(* Logix 5000 project; controller cal1615 1756-L62 rev 20.19; software revision 20.05; part 53 of 82 *)
(* tags used below, declared in another part *)
   p23r17 : routine;
   FAULT : BOOL;   // Fault AFI
   HMI : BOOL;   // AFI HMI
   p01_param_oven_timer_presets : DINT[32];   // System Parameter Oven Timer Presets
   p01r09 : routine;   // System Modes
   p01r09_pb_global_reset : BOOL;   // System Modes PB: Global Fault Reset
   p01r11 : routine;   // System Timer Presets
   p01r13_line_running : BOOL;   // System Line Start Sequence Line Running
   p02_dint_from_hmi : hmi_dint;
   p02_real_from_hmi : hmi_real;   // MOP HMI Iface Real from HMI
   p23_ai_os_masked_gap : REAL;
   p23_ao_servo_os_zero_offset : REAL;   // Impreg Analog Outputs Drive Operator Side Servo Position Offset
   p23_di_servo_os : servo_di;   // Impreg Digital Inputs Servo Operator Side
   p23_di_vfd_jog_fwd : BOOL;   // Impreg Input PB: VFD Jog FWD
   p23_di_vfd_jog_rev : BOOL;   // Impreg Input PB: VFD Jog REV
   p23_dint_to_hmi : DINT[17];   // Impreg Dint to HMI
   p23_do_servo_os : servo_do;   // Impreg Digital Outputs Operator Side Servo
   p23_param_lfl_hhl : REAL;   // Impreg Parameter LFL High High Limit
   p23_param_lfl_hl : REAL;   // Impreg Parameters LFL High Limit
   p23_param_servo_open_position : REAL;
   p23_param_zone_pressure : REAL;   // MOP HMI Iface Parameters Minimum Pressure
   p23r01 : routine;   // Impreg Main
   p23r02 : routine;   // Impreg Misc Control
   p23r08 : routine;   // Impreg Warnings
   p23r08_timer_fault : TIMER[4];   // Impreg Warnings Fault Delay
   p23r08_timer_warning : TIMER[4];   // Impreg Warnings Warning Delay
   p23r09 : routine;   // Impreg Mode Selection
   p23r09_mode_run : BOOL;   // Impreg Modes Pick Up Roll Run Mode
   p23r09_timer_fault : TIMER[4];   // Impreg Mode Selection Fault Delay
   p23r09_web_wet_ctrl_toggle : SYS_Toggle;   // Impreg Metering Roll VFD Web Wet Control
   p23r10 : routine;
   p23r10_timer_fault : TIMER[4];   // Impreg Parameters Fault Dwell Timer
   p23r10_timer_warning : TIMER[4];   // Impreg Parameters Warning Dwell Timer
   p23r11 : routine;   // Impreg Servo Operator Side
   p23r11_gap_sequence_enabled : BOOL;
   p23r11_impreg_gap_os : REAL;
   p23r11_offsets : REAL[100];
   p23r11_permissive_jog : BOOL;   // Impreg Servo Operator Side Perimssive Jog
   p23r11_pos_offset : REAL;
   p23r11_request_jog_fwd : BOOL;   // Impreg Servo Operator Side Requset Jog Forward
   p23r11_request_jog_rev : BOOL;   // Impreg Servo Operator Side Requset Jog Reverse
   p23r11_request_position : BOOL;   // Impreg Servo Operator Side Request Position
   p23r11_request_start : BOOL;   // Impreg Servo Operator Side Request Start
   p23r11_request_zero : BOOL;   // Impreg Servo Operator Side Request Zero
   p23r11_selected_position : REAL;
   p23r11_servo_not_ready : BOOL;   // Impreg Servo Operator Side Not Ready
   p23r11_servo_status_ab : BOOL;   // Impreg Servo Operator Side AB Status
   p23r11_servo_status_af : BOOL;   // Impreg Servo Operator Side AF Status
   p23r11_servo_status_bb : BOOL;   // Impreg Servo Operator Side BB Status
   p23r11_step_4_dwell : TIMER;
   p23r11_timer : TIMER[4];   // Impreg Servo Operator Side Timer
   p23r12 : routine;   // Impreg Servo Drive Side
   p23r13 : routine;
   p23r15 : routine;   // Impreg Metering Roll VFD
   p23r15_pid_tension_control : BOOL;   // Impreg Metering Roll VFD PID Wet Web Active
(* P23_Impreg, continued *)

ROUTINE R08_Warnings   (* ladder *)
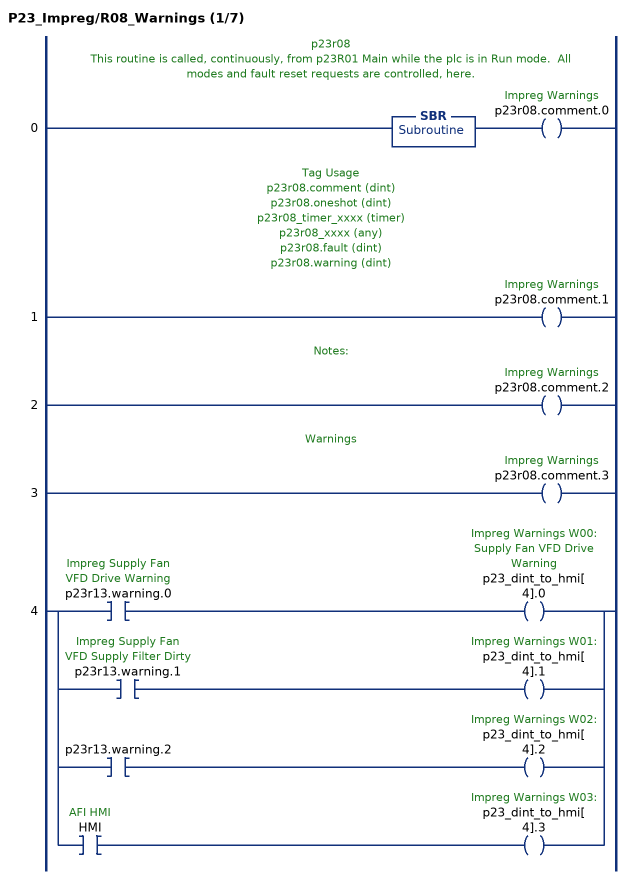
   // p23r08
   // This routine is called, continuously, from p23R01 Main while the plc is in Run mode.  All modes and fault reset requests are controlled, here.
   0: SBR()OTE(p23r08.comment.0);
   // Tag Usage
   // p23r08.comment (dint)
   // p23r08.oneshot (dint)
   // p23r08_timer_xxxx (timer)
   // p23r08_xxxx (any)
   // p23r08.fault (dint)
   // p23r08.warning (dint)
   1: OTE(p23r08.comment.1);
   // Notes:
   2: OTE(p23r08.comment.2);
   // Warnings
   3: OTE(p23r08.comment.3);
   4: [XIC(p23r13.warning.0) OTE(p23_dint_to_hmi[4].0) ,XIC(p23r13.warning.1) OTE(p23_dint_to_hmi[4].1) ,XIC(p23r13.warning.2) OTE(p23_dint_to_hmi[4].2) ,XIC(HMI) OTE(p23_dint_to_hmi[4].3) ];
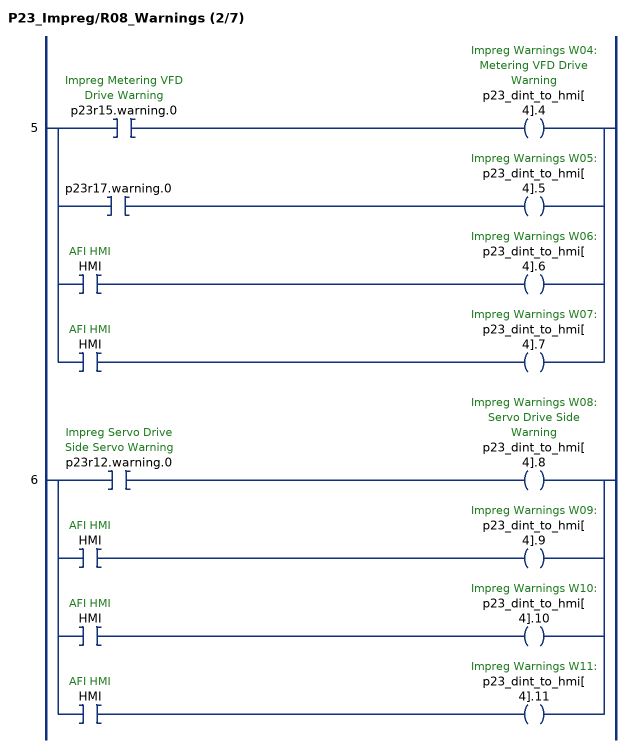
   5: [XIC(p23r15.warning.0) OTE(p23_dint_to_hmi[4].4) ,XIC(p23r17.warning.0) OTE(p23_dint_to_hmi[4].5) ,XIC(HMI) OTE(p23_dint_to_hmi[4].6) ,XIC(HMI) OTE(p23_dint_to_hmi[4].7) ];
   6: [XIC(p23r12.warning.0) OTE(p23_dint_to_hmi[4].8) ,XIC(HMI) OTE(p23_dint_to_hmi[4].9) ,XIC(HMI) OTE(p23_dint_to_hmi[4].10) ,XIC(HMI) OTE(p23_dint_to_hmi[4].11) ];
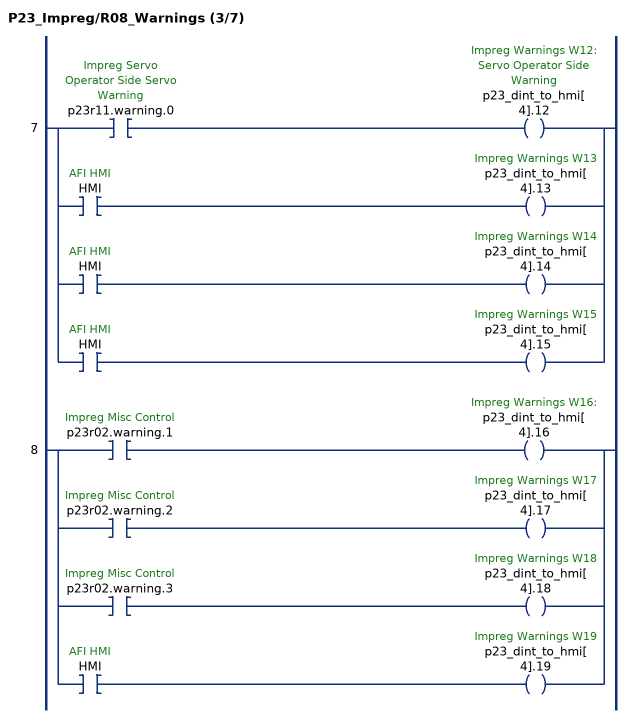
   7: [XIC(p23r11.warning.0) OTE(p23_dint_to_hmi[4].12) ,XIC(HMI) OTE(p23_dint_to_hmi[4].13) ,XIC(HMI) OTE(p23_dint_to_hmi[4].14) ,XIC(HMI) OTE(p23_dint_to_hmi[4].15) ];
   8: [XIC(p23r02.warning.1) OTE(p23_dint_to_hmi[4].16) ,XIC(p23r02.warning.2) OTE(p23_dint_to_hmi[4].17) ,XIC(p23r02.warning.3) OTE(p23_dint_to_hmi[4].18) ,XIC(HMI) OTE(p23_dint_to_hmi[4].19) ];
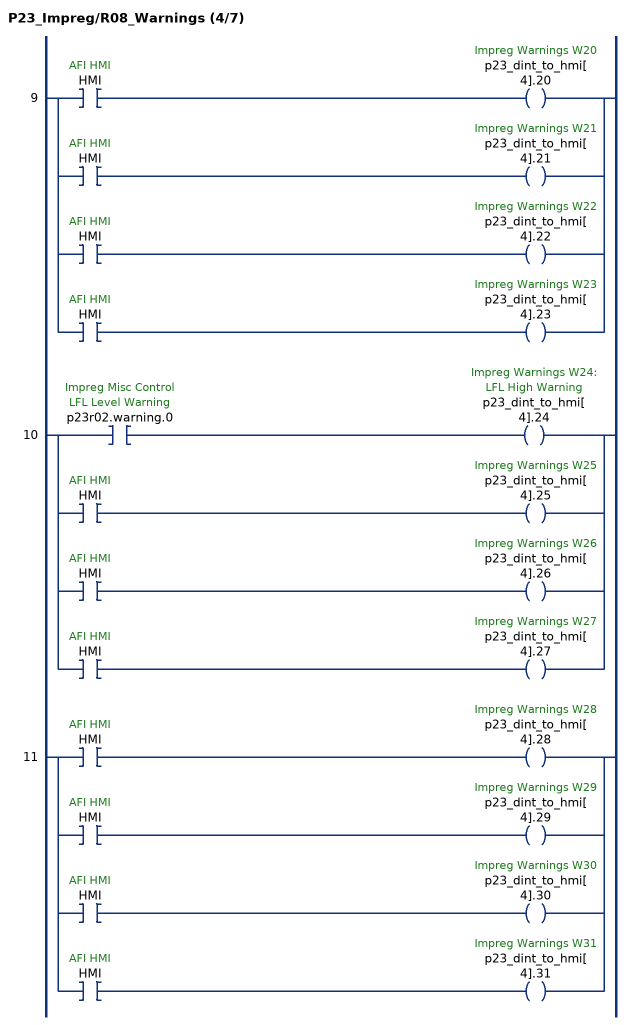
   9: [XIC(HMI) OTE(p23_dint_to_hmi[4].20) ,XIC(HMI) OTE(p23_dint_to_hmi[4].21) ,XIC(HMI) OTE(p23_dint_to_hmi[4].22) ,XIC(HMI) OTE(p23_dint_to_hmi[4].23) ];
   10: [XIC(p23r02.warning.0) OTE(p23_dint_to_hmi[4].24) ,XIC(HMI) OTE(p23_dint_to_hmi[4].25) ,XIC(HMI) OTE(p23_dint_to_hmi[4].26) ,XIC(HMI) OTE(p23_dint_to_hmi[4].27) ];
   11: [XIC(HMI) OTE(p23_dint_to_hmi[4].28) ,XIC(HMI) OTE(p23_dint_to_hmi[4].29) ,XIC(HMI) OTE(p23_dint_to_hmi[4].30) ,XIC(HMI) OTE(p23_dint_to_hmi[4].31) ];
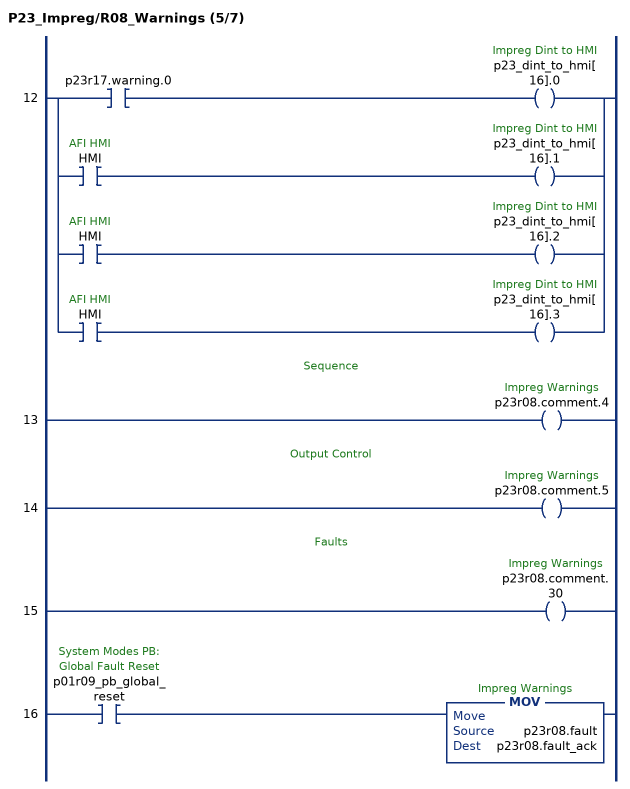
   12: [XIC(p23r17.warning.0) OTE(p23_dint_to_hmi[16].0) ,XIC(HMI) OTE(p23_dint_to_hmi[16].1) ,XIC(HMI) OTE(p23_dint_to_hmi[16].2) ,XIC(HMI) OTE(p23_dint_to_hmi[16].3) ];
   // Sequence
   13: OTE(p23r08.comment.4);
   // Output Control
   14: OTE(p23r08.comment.5);
   // Faults
   15: OTE(p23r08.comment.30);
   16: XIC(p01r09_pb_global_reset)MOV(p23r08.fault,p23r08.fault_ack);
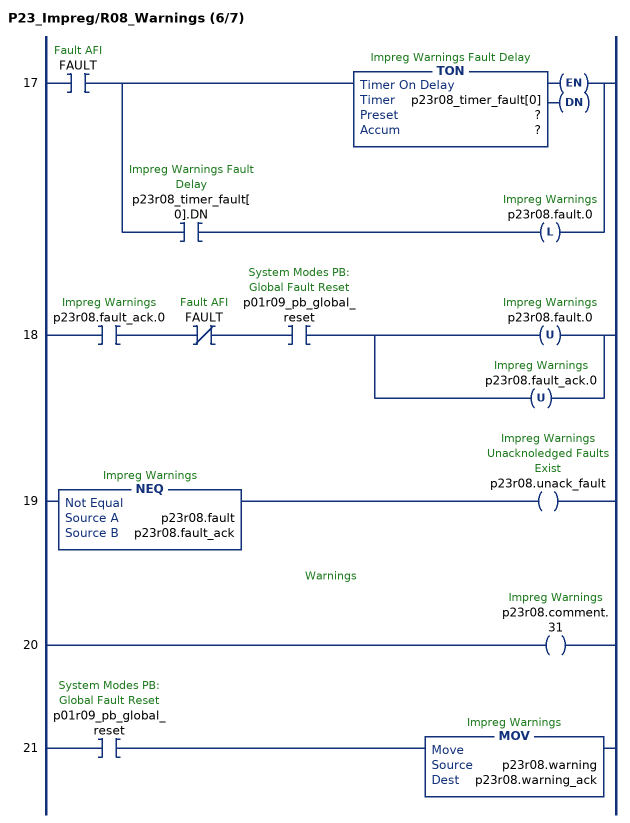
   17: XIC(FAULT)[TON(p23r08_timer_fault[0],?,?) ,XIC(p23r08_timer_fault[0].DN) OTL(p23r08.fault.0) ];
   18: XIC(p23r08.fault_ack.0)XIO(FAULT)XIC(p01r09_pb_global_reset)[OTU(p23r08.fault.0) ,OTU(p23r08.fault_ack.0) ];
   19: NEQ(p23r08.fault,p23r08.fault_ack)OTE(p23r08.unack_fault);
   // Warnings
   20: OTE(p23r08.comment.31);
   21: XIC(p01r09_pb_global_reset)MOV(p23r08.warning,p23r08.warning_ack);
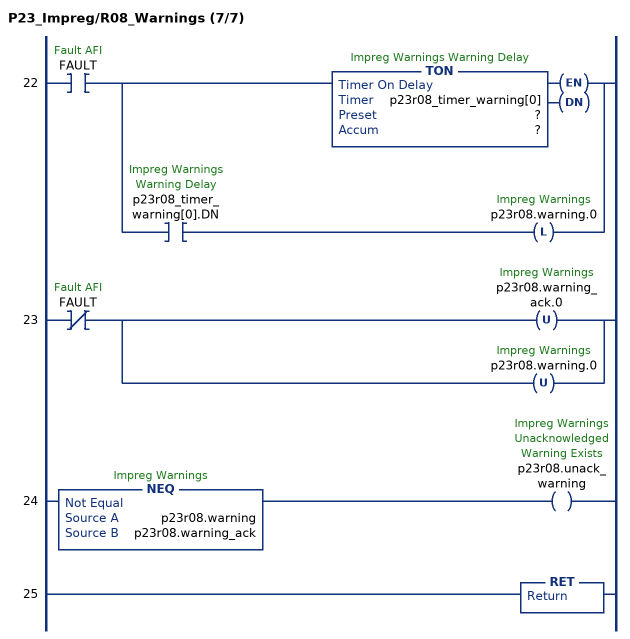
   22: XIC(FAULT)[TON(p23r08_timer_warning[0],?,?) ,XIC(p23r08_timer_warning[0].DN) OTL(p23r08.warning.0) ];
   23: XIO(FAULT)[OTU(p23r08.warning_ack.0) ,OTU(p23r08.warning.0) ];
   24: NEQ(p23r08.warning,p23r08.warning_ack)OTE(p23r08.unack_warning);
   25: RET();
END_ROUTINE

ROUTINE R09_Modes   (* ladder *)
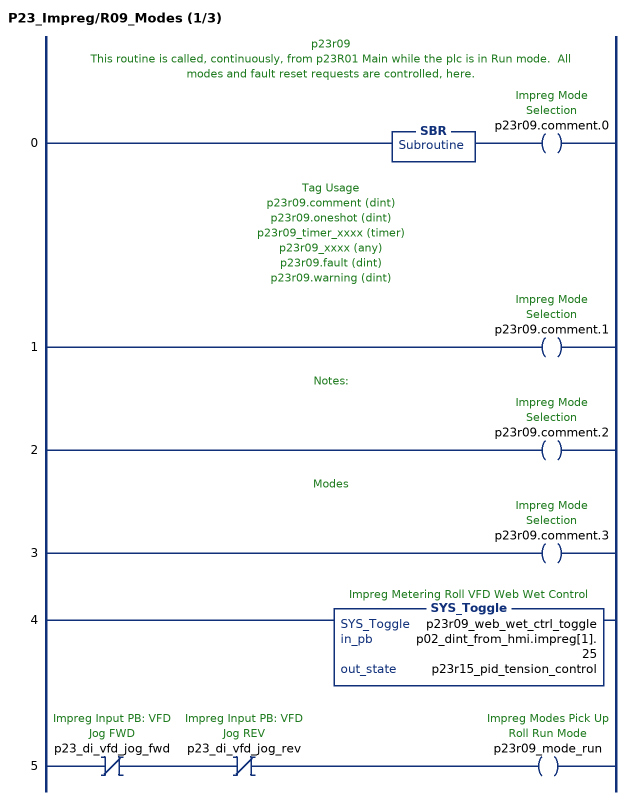
   // p23r09
   // This routine is called, continuously, from p23R01 Main while the plc is in Run mode.  All modes and fault reset requests are controlled, here.
   0: SBR()OTE(p23r09.comment.0);
   // Tag Usage
   // p23r09.comment (dint)
   // p23r09.oneshot (dint)
   // p23r09_timer_xxxx (timer)
   // p23r09_xxxx (any)
   // p23r09.fault (dint)
   // p23r09.warning (dint)
   1: OTE(p23r09.comment.1);
   // Notes:
   2: OTE(p23r09.comment.2);
   // Modes
   3: OTE(p23r09.comment.3);
   4: SYS_Toggle(p23r09_web_wet_ctrl_toggle,p02_dint_from_hmi.impreg[1].25,p23r15_pid_tension_control);
   5: XIO(p23_di_vfd_jog_fwd)XIO(p23_di_vfd_jog_rev)OTE(p23r09_mode_run);
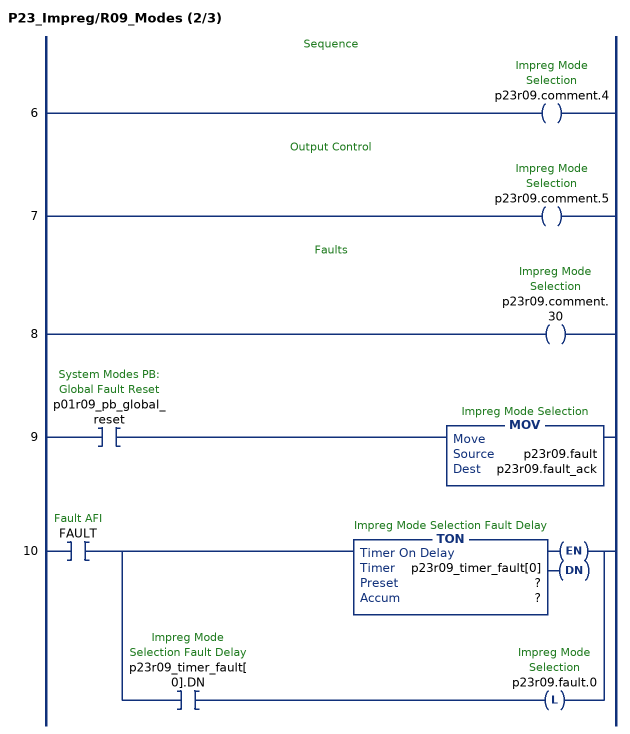
   // Sequence
   6: OTE(p23r09.comment.4);
   // Output Control
   7: OTE(p23r09.comment.5);
   // Faults
   8: OTE(p23r09.comment.30);
   9: XIC(p01r09_pb_global_reset)MOV(p23r09.fault,p23r09.fault_ack);
   10: XIC(FAULT)[TON(p23r09_timer_fault[0],?,?) ,XIC(p23r09_timer_fault[0].DN) OTL(p23r09.fault.0) ];
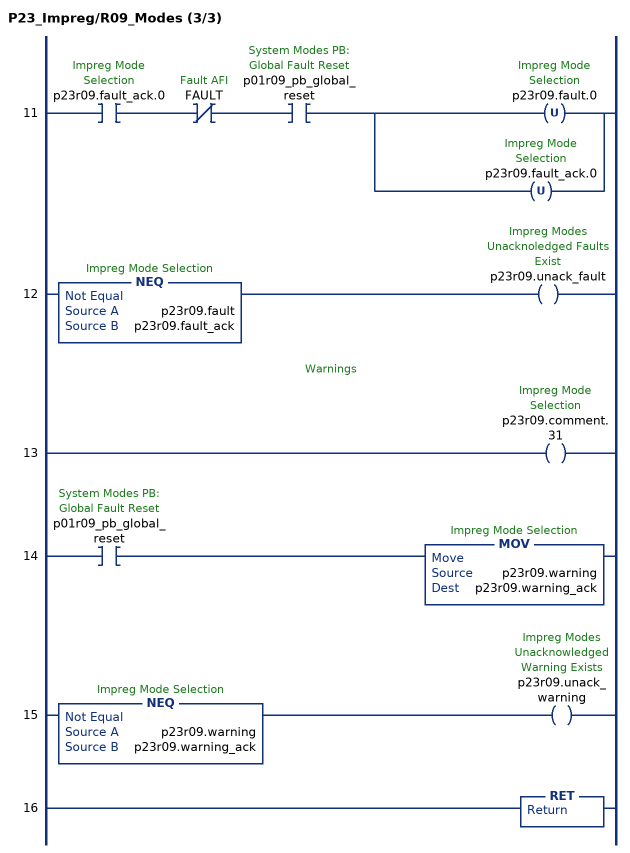
   11: XIC(p23r09.fault_ack.0)XIO(FAULT)XIC(p01r09_pb_global_reset)[OTU(p23r09.fault.0) ,OTU(p23r09.fault_ack.0) ];
   12: NEQ(p23r09.fault,p23r09.fault_ack)OTE(p23r09.unack_fault);
   // Warnings
   13: OTE(p23r09.comment.31);
   14: XIC(p01r09_pb_global_reset)MOV(p23r09.warning,p23r09.warning_ack);
   15: NEQ(p23r09.warning,p23r09.warning_ack)OTE(p23r09.unack_warning);
   16: RET();
END_ROUTINE

ROUTINE R10_Parameters   (* ladder *)
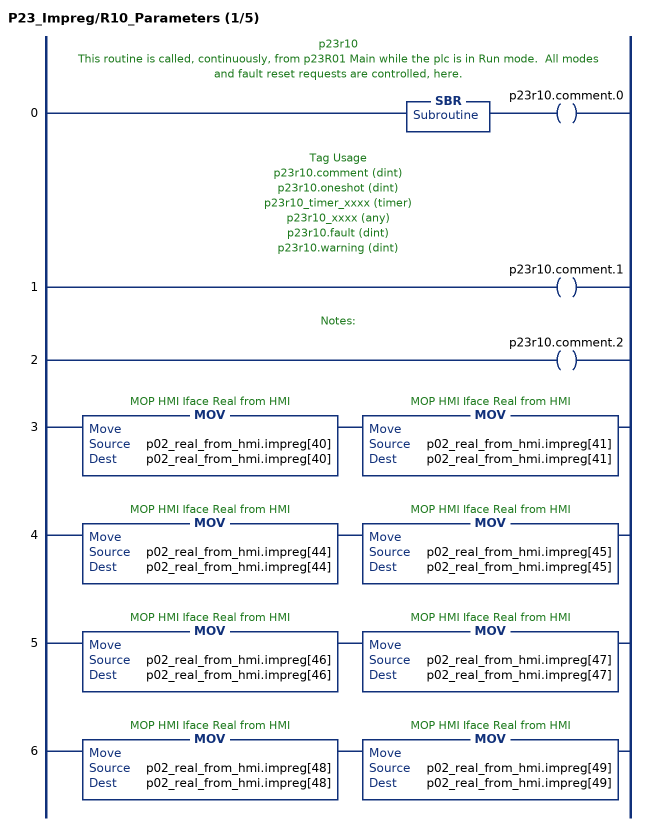
   // p23r10
   // This routine is called, continuously, from p23R01 Main while the plc is in Run mode.  All modes and fault reset requests are controlled, here.
   0: SBR()OTE(p23r10.comment.0);
   // Tag Usage
   // p23r10.comment (dint)
   // p23r10.oneshot (dint)
   // p23r10_timer_xxxx (timer)
   // p23r10_xxxx (any)
   // p23r10.fault (dint)
   // p23r10.warning (dint)
   1: OTE(p23r10.comment.1);
   // Notes:
   2: OTE(p23r10.comment.2);
   3: MOV(p02_real_from_hmi.impreg[40],p02_real_from_hmi.impreg[40])MOV(p02_real_from_hmi.impreg[41],p02_real_from_hmi.impreg[41]);
   4: MOV(p02_real_from_hmi.impreg[44],p02_real_from_hmi.impreg[44])MOV(p02_real_from_hmi.impreg[45],p02_real_from_hmi.impreg[45]);
   5: MOV(p02_real_from_hmi.impreg[46],p02_real_from_hmi.impreg[46])MOV(p02_real_from_hmi.impreg[47],p02_real_from_hmi.impreg[47]);
   6: MOV(p02_real_from_hmi.impreg[48],p02_real_from_hmi.impreg[48])MOV(p02_real_from_hmi.impreg[49],p02_real_from_hmi.impreg[49]);
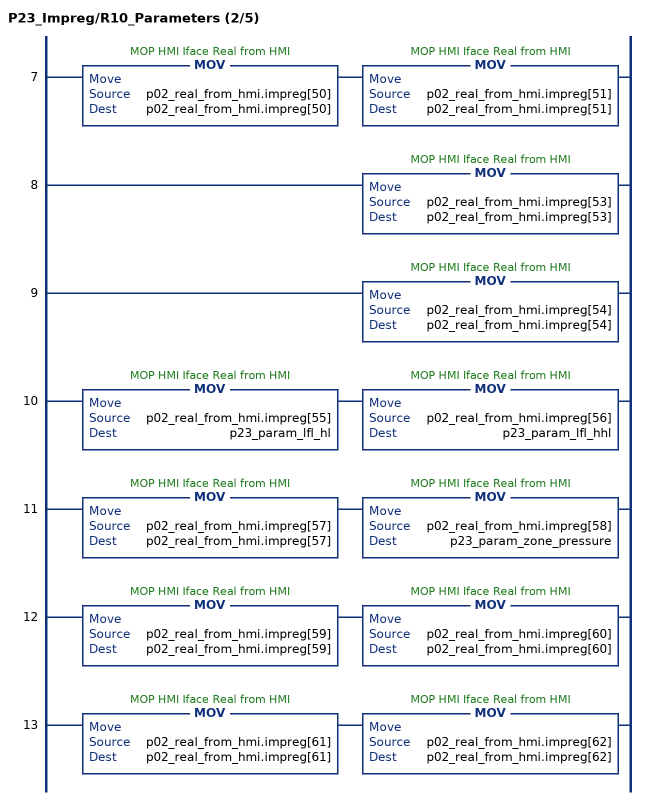
   7: MOV(p02_real_from_hmi.impreg[50],p02_real_from_hmi.impreg[50])MOV(p02_real_from_hmi.impreg[51],p02_real_from_hmi.impreg[51]);
   8: MOV(p02_real_from_hmi.impreg[53],p02_real_from_hmi.impreg[53]);
   9: MOV(p02_real_from_hmi.impreg[54],p02_real_from_hmi.impreg[54]);
   10: MOV(p02_real_from_hmi.impreg[55],p23_param_lfl_hl)MOV(p02_real_from_hmi.impreg[56],p23_param_lfl_hhl);
   11: MOV(p02_real_from_hmi.impreg[57],p02_real_from_hmi.impreg[57])MOV(p02_real_from_hmi.impreg[58],p23_param_zone_pressure);
   12: MOV(p02_real_from_hmi.impreg[59],p02_real_from_hmi.impreg[59])MOV(p02_real_from_hmi.impreg[60],p02_real_from_hmi.impreg[60]);
   13: MOV(p02_real_from_hmi.impreg[61],p02_real_from_hmi.impreg[61])MOV(p02_real_from_hmi.impreg[62],p02_real_from_hmi.impreg[62]);
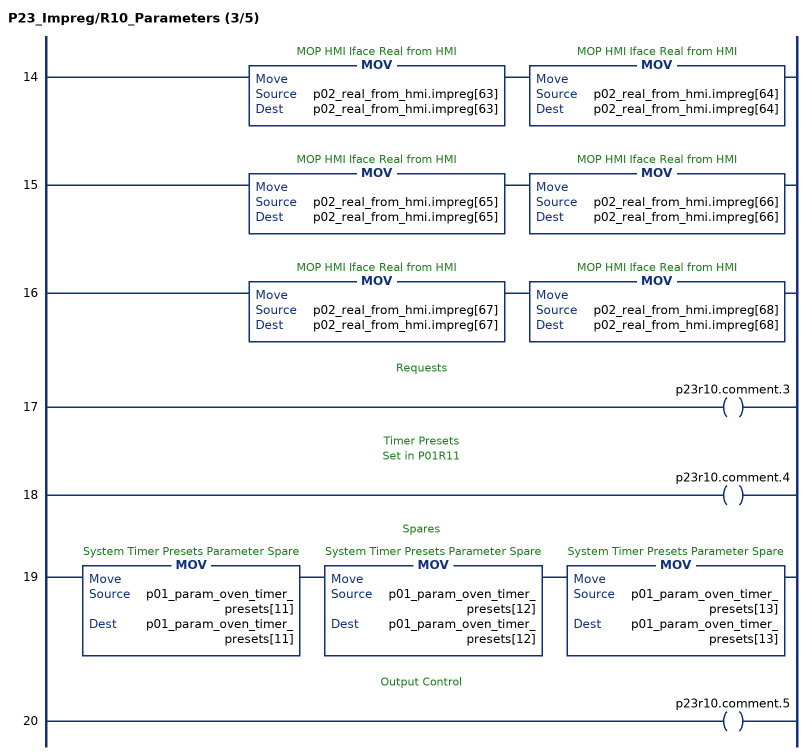
   14: MOV(p02_real_from_hmi.impreg[63],p02_real_from_hmi.impreg[63])MOV(p02_real_from_hmi.impreg[64],p02_real_from_hmi.impreg[64]);
   15: MOV(p02_real_from_hmi.impreg[65],p02_real_from_hmi.impreg[65])MOV(p02_real_from_hmi.impreg[66],p02_real_from_hmi.impreg[66]);
   16: MOV(p02_real_from_hmi.impreg[67],p02_real_from_hmi.impreg[67])MOV(p02_real_from_hmi.impreg[68],p02_real_from_hmi.impreg[68]);
   // Requests
   17: OTE(p23r10.comment.3);
   // Timer Presets
   // Set in P01R11
   18: OTE(p23r10.comment.4);
   // Spares
   19: MOV(p01_param_oven_timer_presets[11],p01_param_oven_timer_presets[11])MOV(p01_param_oven_timer_presets[12],p01_param_oven_timer_presets[12])MOV(p01_param_oven_timer_presets[13],p01_param_oven_timer_presets[13]);
   // Output Control
   20: OTE(p23r10.comment.5);
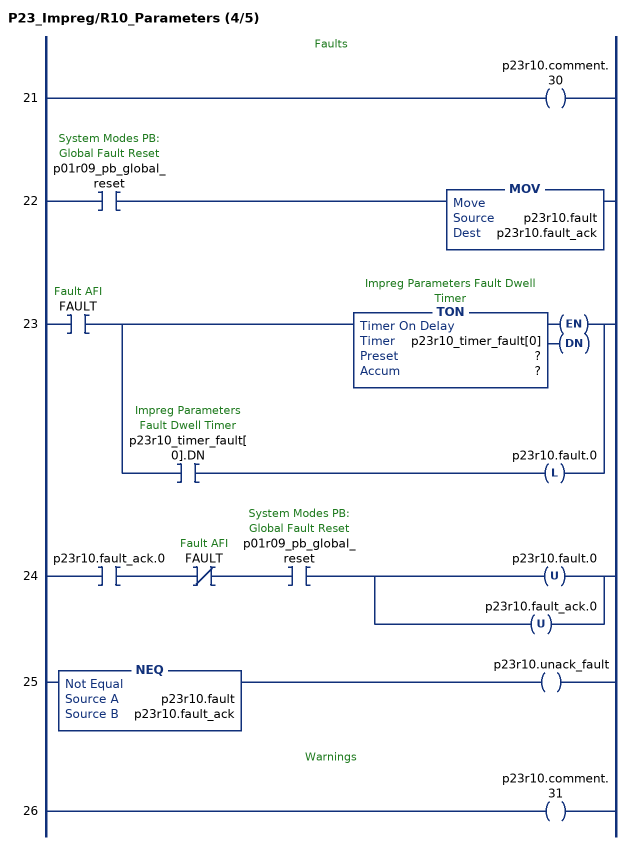
   // Faults
   21: OTE(p23r10.comment.30);
   22: XIC(p01r09_pb_global_reset)MOV(p23r10.fault,p23r10.fault_ack);
   23: XIC(FAULT)[TON(p23r10_timer_fault[0],?,?) ,XIC(p23r10_timer_fault[0].DN) OTL(p23r10.fault.0) ];
   24: XIC(p23r10.fault_ack.0)XIO(FAULT)XIC(p01r09_pb_global_reset)[OTU(p23r10.fault.0) ,OTU(p23r10.fault_ack.0) ];
   25: NEQ(p23r10.fault,p23r10.fault_ack)OTE(p23r10.unack_fault);
   // Warnings
   26: OTE(p23r10.comment.31);
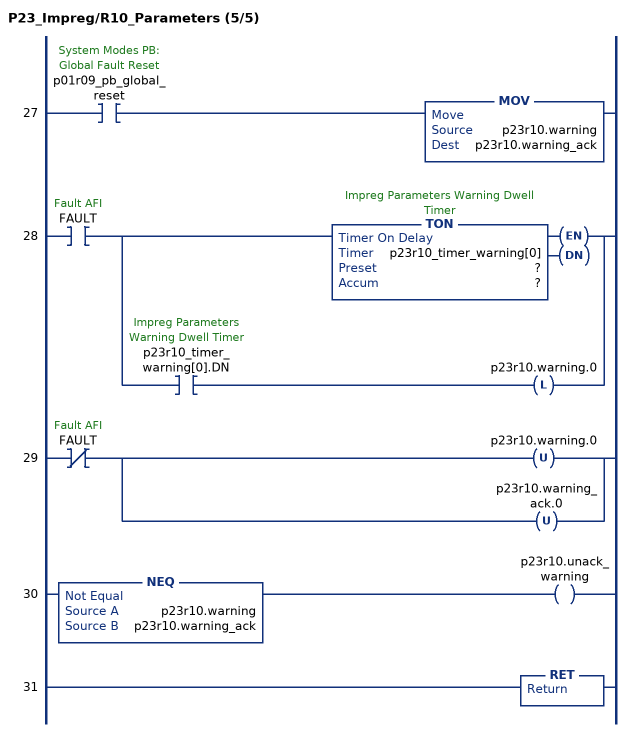
   27: XIC(p01r09_pb_global_reset)MOV(p23r10.warning,p23r10.warning_ack);
   28: XIC(FAULT)[TON(p23r10_timer_warning[0],?,?) ,XIC(p23r10_timer_warning[0].DN) OTL(p23r10.warning.0) ];
   29: XIO(FAULT)[OTU(p23r10.warning.0) ,OTU(p23r10.warning_ack.0) ];
   30: NEQ(p23r10.warning,p23r10.warning_ack)OTE(p23r10.unack_warning);
   31: RET();
END_ROUTINE

ROUTINE R11_Servo_Operator_Side   (* ladder *)
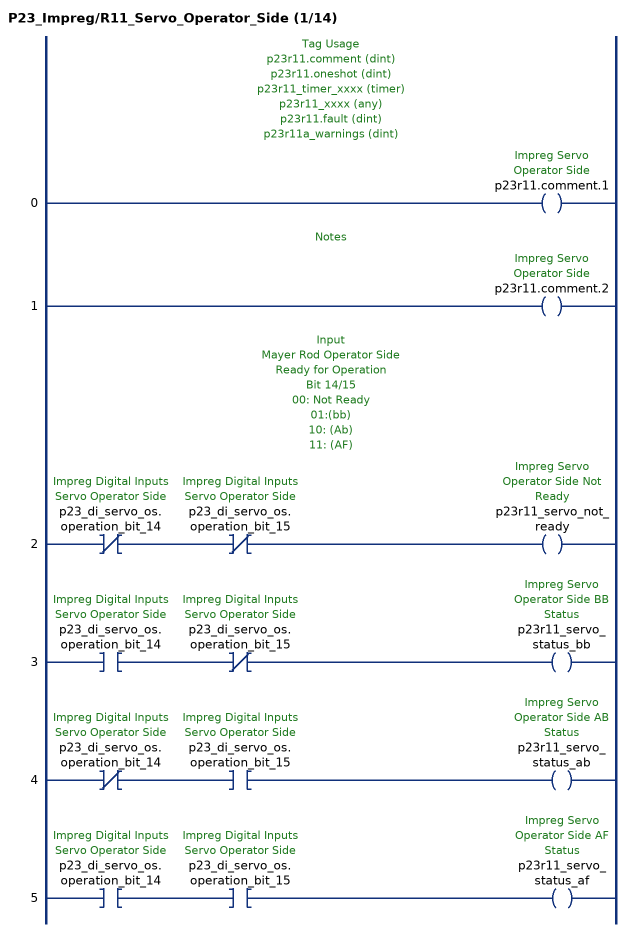
   // Tag Usage
   // p23r11.comment (dint)
   // p23r11.oneshot (dint)
   // p23r11_timer_xxxx (timer)
   // p23r11_xxxx (any)
   // p23r11.fault (dint)
   // p23r11a_warnings (dint)
   0: OTE(p23r11.comment.1);
   // Notes
   1: OTE(p23r11.comment.2);
   // Input
   // Mayer Rod Operator Side
   // Ready for Operation
   // Bit 14/15
   // 00: Not Ready
   // 01:(bb)
   // 10: (Ab)
   // 11: (AF)
   2: XIO(p23_di_servo_os.operation_bit_14)XIO(p23_di_servo_os.operation_bit_15)OTE(p23r11_servo_not_ready);
   3: XIC(p23_di_servo_os.operation_bit_14)XIO(p23_di_servo_os.operation_bit_15)OTE(p23r11_servo_status_bb);
   4: XIO(p23_di_servo_os.operation_bit_14)XIC(p23_di_servo_os.operation_bit_15)OTE(p23r11_servo_status_ab);
   5: XIC(p23_di_servo_os.operation_bit_14)XIC(p23_di_servo_os.operation_bit_15)OTE(p23r11_servo_status_af);
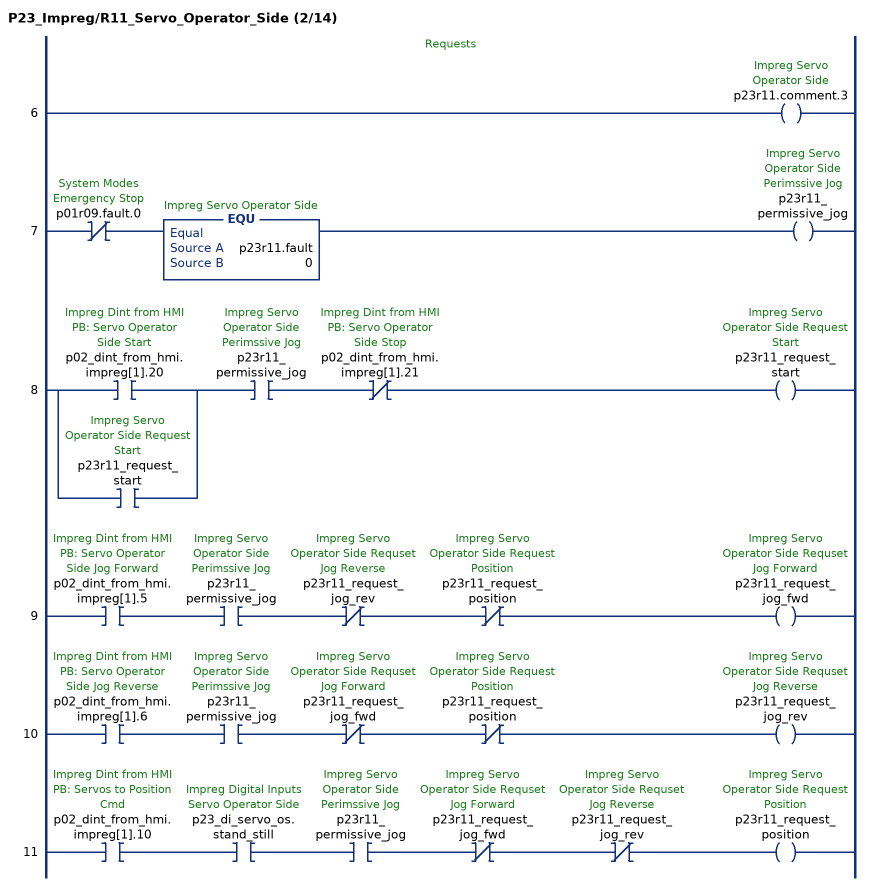
   // Requests
   6: OTE(p23r11.comment.3);
   7: XIO(p01r09.fault.0)EQU(p23r11.fault,0)OTE(p23r11_permissive_jog);
   8: [XIC(p02_dint_from_hmi.impreg[1].20) ,XIC(p23r11_request_start) ]XIC(p23r11_permissive_jog)XIO(p02_dint_from_hmi.impreg[1].21)OTE(p23r11_request_start);
   9: XIC(p02_dint_from_hmi.impreg[1].5)XIC(p23r11_permissive_jog)XIO(p23r11_request_jog_rev)XIO(p23r11_request_position)OTE(p23r11_request_jog_fwd);
   10: XIC(p02_dint_from_hmi.impreg[1].6)XIC(p23r11_permissive_jog)XIO(p23r11_request_jog_fwd)XIO(p23r11_request_position)OTE(p23r11_request_jog_rev);
   11: XIC(p02_dint_from_hmi.impreg[1].10)XIC(p23_di_servo_os.stand_still)XIC(p23r11_permissive_jog)XIO(p23r11_request_jog_fwd)XIO(p23r11_request_jog_rev)OTE(p23r11_request_position);
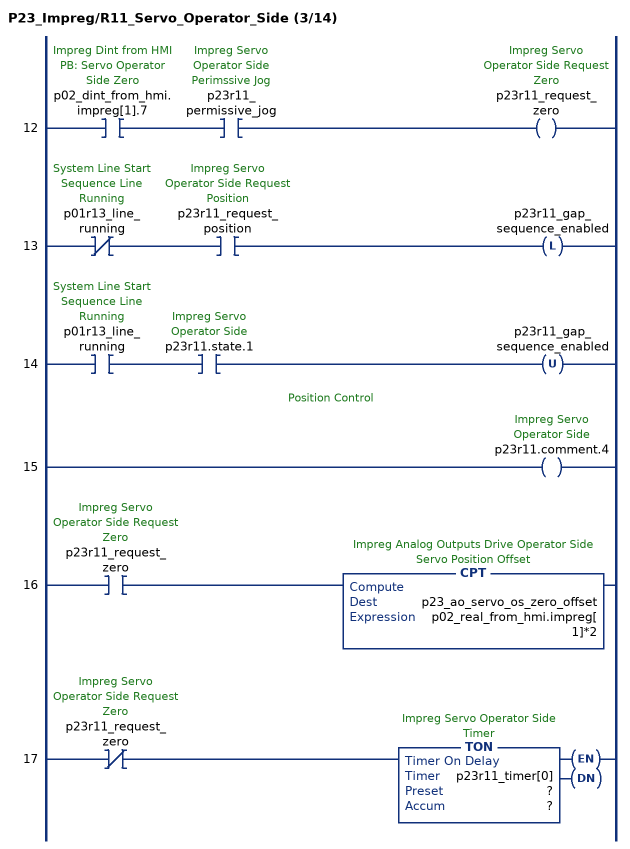
   12: XIC(p02_dint_from_hmi.impreg[1].7)XIC(p23r11_permissive_jog)OTE(p23r11_request_zero);
   13: XIO(p01r13_line_running)XIC(p23r11_request_position)OTL(p23r11_gap_sequence_enabled);
   14: XIC(p01r13_line_running)XIC(p23r11.state.1)OTU(p23r11_gap_sequence_enabled);
   // Position Control
   15: OTE(p23r11.comment.4);
   16: XIC(p23r11_request_zero)CPT(p23_ao_servo_os_zero_offset,p02_real_from_hmi.impreg[1]*2);
   17: XIO(p23r11_request_zero)TON(p23r11_timer[0],?,?);
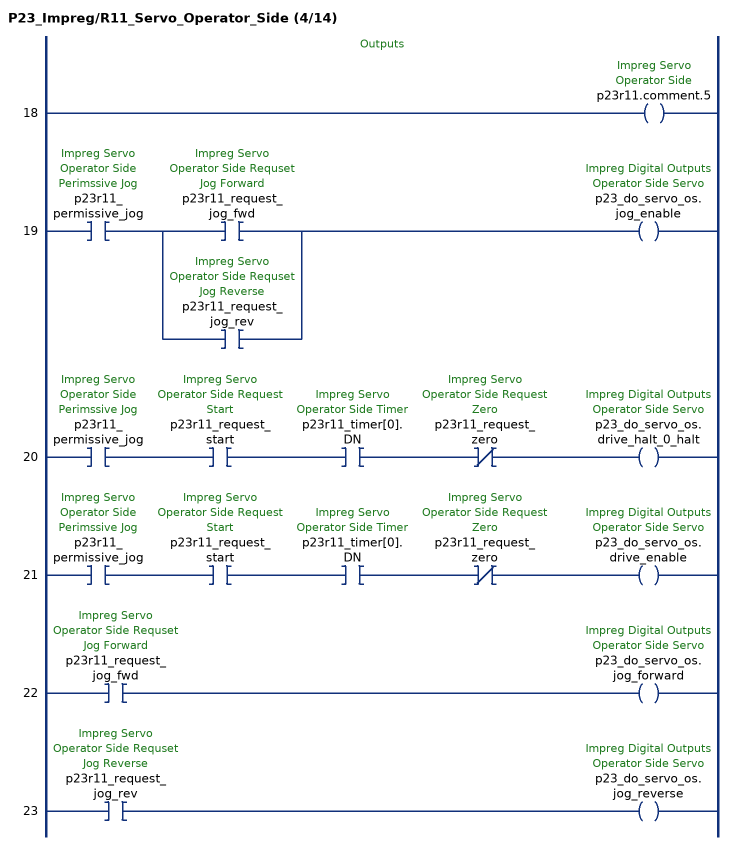
   // Outputs
   18: OTE(p23r11.comment.5);
   19: XIC(p23r11_permissive_jog)[XIC(p23r11_request_jog_fwd) ,XIC(p23r11_request_jog_rev) ]OTE(p23_do_servo_os.jog_enable);
   20: XIC(p23r11_permissive_jog)XIC(p23r11_request_start)XIC(p23r11_timer[0].DN)XIO(p23r11_request_zero)OTE(p23_do_servo_os.drive_halt_0_halt);
   21: XIC(p23r11_permissive_jog)XIC(p23r11_request_start)XIC(p23r11_timer[0].DN)XIO(p23r11_request_zero)OTE(p23_do_servo_os.drive_enable);
   22: XIC(p23r11_request_jog_fwd)OTE(p23_do_servo_os.jog_forward);
   23: XIC(p23r11_request_jog_rev)OTE(p23_do_servo_os.jog_reverse);
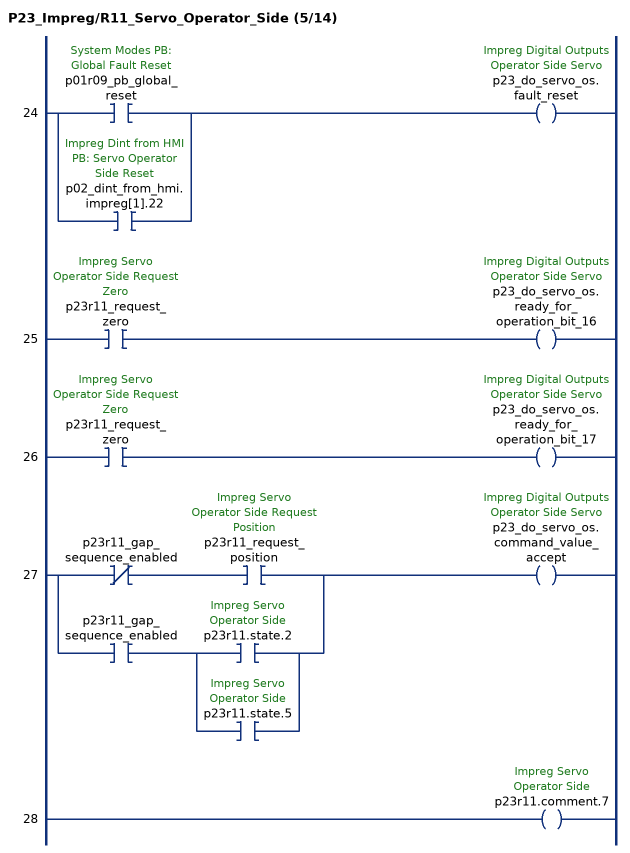
   24: [XIC(p01r09_pb_global_reset) ,XIC(p02_dint_from_hmi.impreg[1].22) ]OTE(p23_do_servo_os.fault_reset);
   25: XIC(p23r11_request_zero)OTE(p23_do_servo_os.ready_for_operation_bit_16);
   26: XIC(p23r11_request_zero)OTE(p23_do_servo_os.ready_for_operation_bit_17);
   27: [XIO(p23r11_gap_sequence_enabled) XIC(p23r11_request_position) ,XIC(p23r11_gap_sequence_enabled) [XIC(p23r11.state.2) ,XIC(p23r11.state.5) ] ]OTE(p23_do_servo_os.command_value_accept);
   28: OTE(p23r11.comment.7);
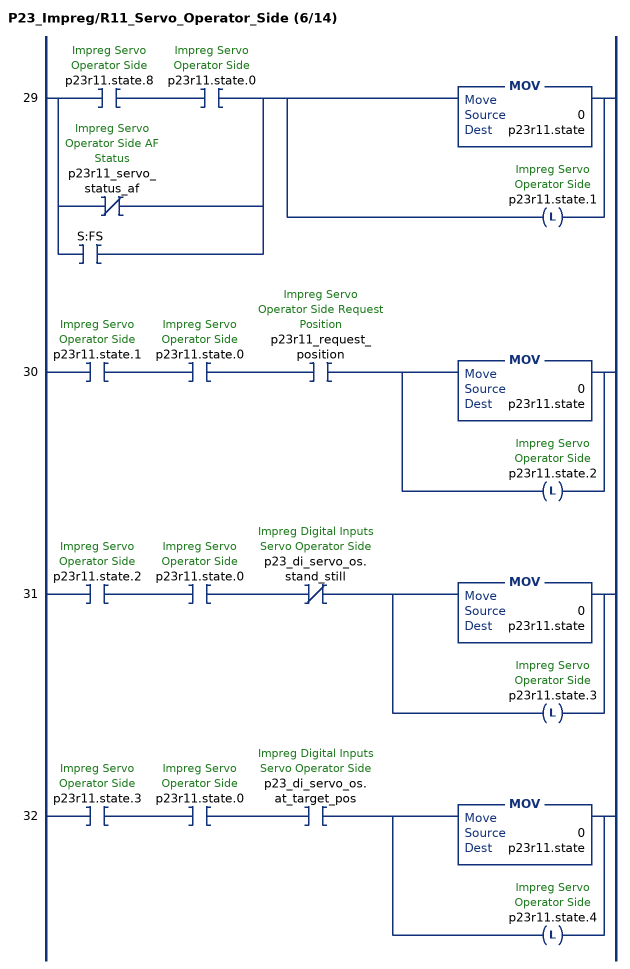
   29: [XIC(p23r11.state.8) XIC(p23r11.state.0) ,XIO(p23r11_servo_status_af) ,XIC(S:FS) ][MOV(0,p23r11.state) ,OTL(p23r11.state.1) ];
   30: XIC(p23r11.state.1)XIC(p23r11.state.0)XIC(p23r11_request_position)[MOV(0,p23r11.state) ,OTL(p23r11.state.2) ];
   31: XIC(p23r11.state.2)XIC(p23r11.state.0)XIO(p23_di_servo_os.stand_still)[MOV(0,p23r11.state) ,OTL(p23r11.state.3) ];
   32: XIC(p23r11.state.3)XIC(p23r11.state.0)XIC(p23_di_servo_os.at_target_pos)[MOV(0,p23r11.state) ,OTL(p23r11.state.4) ];
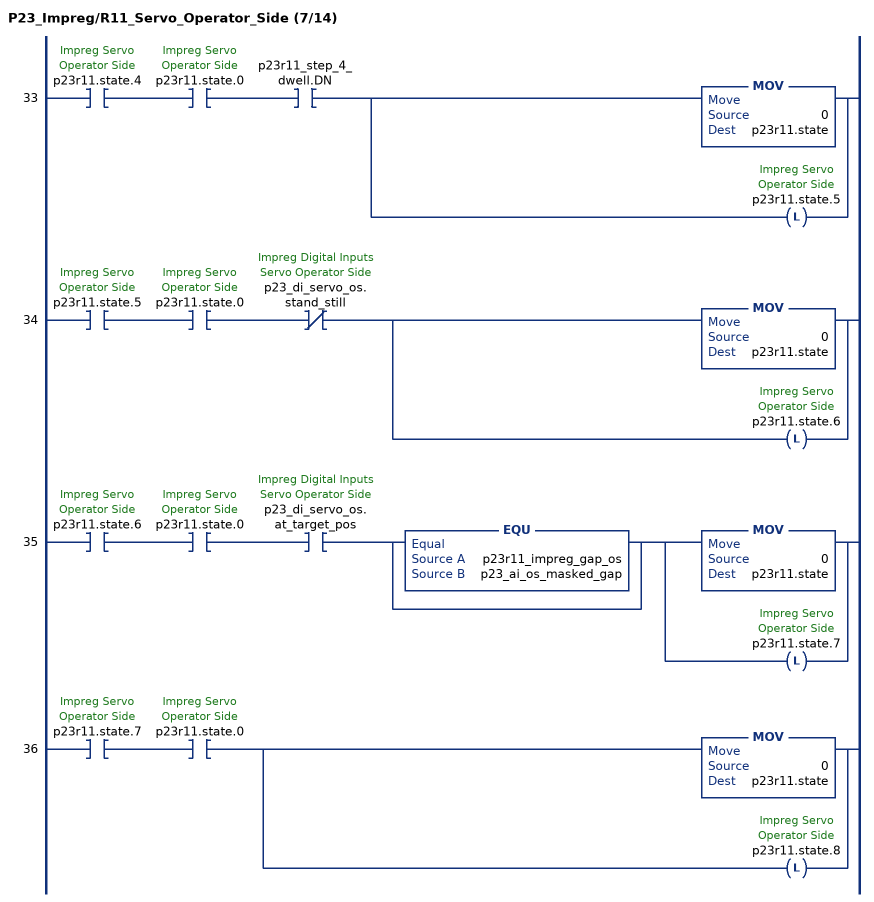
   33: XIC(p23r11.state.4)XIC(p23r11.state.0)XIC(p23r11_step_4_dwell.DN)[MOV(0,p23r11.state) ,OTL(p23r11.state.5) ];
   34: XIC(p23r11.state.5)XIC(p23r11.state.0)XIO(p23_di_servo_os.stand_still)[MOV(0,p23r11.state) ,OTL(p23r11.state.6) ];
   35: XIC(p23r11.state.6)XIC(p23r11.state.0)XIC(p23_di_servo_os.at_target_pos)[EQU(p23r11_impreg_gap_os,p23_ai_os_masked_gap) ,][MOV(0,p23r11.state) ,OTL(p23r11.state.7) ];
   36: XIC(p23r11.state.7)XIC(p23r11.state.0)[MOV(0,p23r11.state) ,OTL(p23r11.state.8) ];
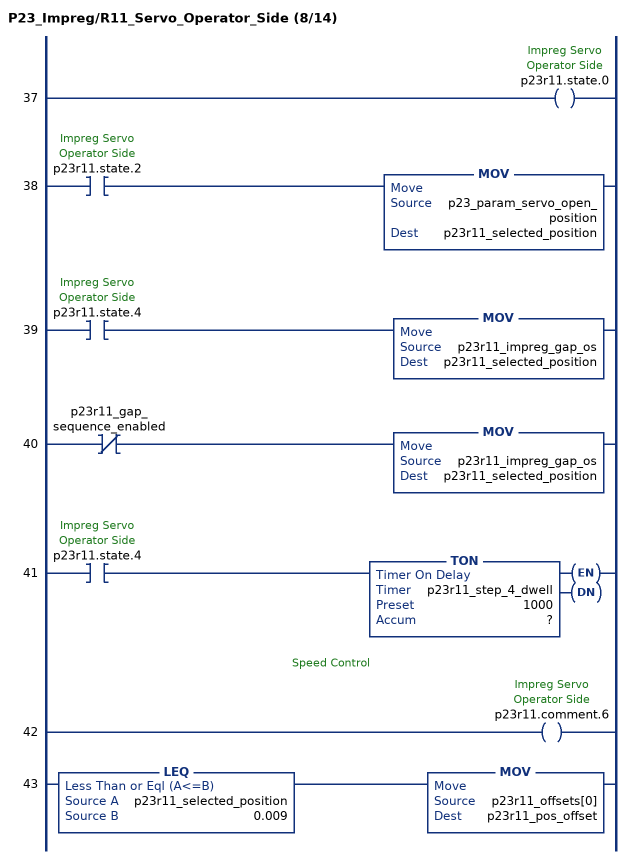
   37: OTE(p23r11.state.0);
   38: XIC(p23r11.state.2)MOV(p23_param_servo_open_position,p23r11_selected_position);
   39: XIC(p23r11.state.4)MOV(p23r11_impreg_gap_os,p23r11_selected_position);
   40: XIO(p23r11_gap_sequence_enabled)MOV(p23r11_impreg_gap_os,p23r11_selected_position);
   41: XIC(p23r11.state.4)TON(p23r11_step_4_dwell,?,?);
   // Speed Control
   42: OTE(p23r11.comment.6);
   43: LEQ(p23r11_selected_position,0.009)MOV(p23r11_offsets[0],p23r11_pos_offset);
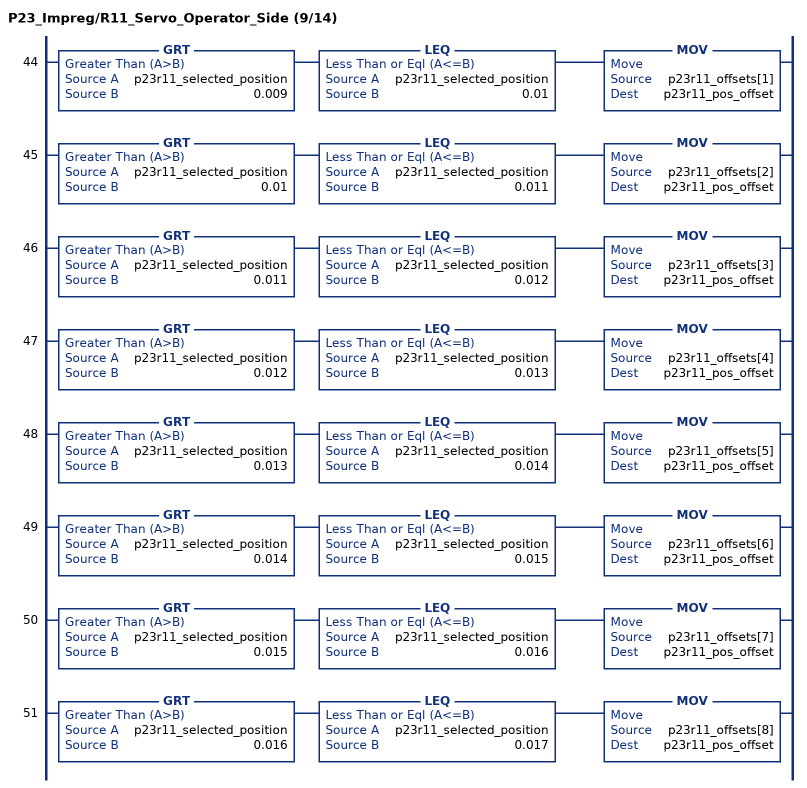
   44: GRT(p23r11_selected_position,0.009)LEQ(p23r11_selected_position,0.01)MOV(p23r11_offsets[1],p23r11_pos_offset);
   45: GRT(p23r11_selected_position,0.01)LEQ(p23r11_selected_position,0.011)MOV(p23r11_offsets[2],p23r11_pos_offset);
   46: GRT(p23r11_selected_position,0.011)LEQ(p23r11_selected_position,0.012)MOV(p23r11_offsets[3],p23r11_pos_offset);
   47: GRT(p23r11_selected_position,0.012)LEQ(p23r11_selected_position,0.013)MOV(p23r11_offsets[4],p23r11_pos_offset);
   48: GRT(p23r11_selected_position,0.013)LEQ(p23r11_selected_position,0.014)MOV(p23r11_offsets[5],p23r11_pos_offset);
   49: GRT(p23r11_selected_position,0.014)LEQ(p23r11_selected_position,0.015)MOV(p23r11_offsets[6],p23r11_pos_offset);
   50: GRT(p23r11_selected_position,0.015)LEQ(p23r11_selected_position,0.016)MOV(p23r11_offsets[7],p23r11_pos_offset);
   51: GRT(p23r11_selected_position,0.016)LEQ(p23r11_selected_position,0.017)MOV(p23r11_offsets[8],p23r11_pos_offset);
